PROGRAM FindBundlesFromDB EXTENDS SqldbReadWrite
VAR_INPUT
	id : STRING;
END_VAR
VAR_OUTPUT
	basicBundlesArr : ARRAY[0..20-1] OF BasicBundle;
END_VAR
VAR
	fbSQLCommand : FB_SQLCommandEvt(sNetID := '', tTimeout := T#5S);
	fbSQLDatabase : FB_SQLDatabaseEvt (sNetID := '', tTimeout := T#5S);
	fbSQLResult : FB_SQLResultEvt(sNetID:='', tTimeout:=T#5S);
	
	query : STRING(1000);
	//step : (RESET, CONNECT, IDLE, EXECUTE, LOAD_DATA, DISCONNECT);
END_VAR
VAR
	stringBuilder : StringBuilder;
	i : INT;
END_VAR

IF NOT ready THEN
	setup();
	RETURN;
END_IF

CASE step OF
	(*
	RESET:
		step := DISCONNECT;
		
	CONNECT:
		IF fbSQLDatabase.Connect(1) THEN
			IF NOT fbSqlDatabase.bError THEN
				step := IDLE;
			END_IF
		END_IF
	*)
	IDLE:
		IF fbSQLDatabase.CreateCmd(ADR(fbSQLCommand)) THEN
			step := EXECUTE;
		END_IF
	
	EXECUTE:
		createQuery();
		IF fbSQLCommand.ExecuteDataReturn(ADR(query), SIZEOF(query), ADR(fbSqlResult)) THEN
			step := IDLE;
		END_IF
	
	LOAD_DATA:
		(*
		fbSqlResult.Read(0, 1, ADR(existingID), SIZEOF(existingID), TRUE, FALSE);
		IF BundleData.id = existingID THEN
			bundleExists := TRUE;
		ELSE
			bundleExists := FALSE;
		END_IF
		IF fbSQLDatabase.Disconnect() THEN
			fbSqlResult.Release();
			checkExistingBundles := TRUE;
			dbCheckStep := CONNECT;
		END_IF
		*)
		
	DISCONNECT:
		IF fbSQLDatabase.Disconnect() THEN
			step := CONNECT;
		END_IF
END_CASE

METHOD PRIVATE createQuery : BOOL
IF id = '' THEN //FINISH WITH OTHER BASIC ATTRIBUTES
	CONCAT2(ADR(query), ADR('SELECT BundleID FROM "Bundle Data - Prototype"'), ADR(query), SIZEOF(query));
ELSE
	CONCAT2(ADR(query), ADR('SELECT BundleID FROM "Bundle Data - Prototype" WHERE BundleID = $''), ADR(query), SIZEOF(query));
	CONCAT2(ADR(query), ADR(id), ADR(query), SIZEOF(query));
	CONCAT2(ADR(query), ADR('$''), ADR(query), SIZEOF(query));
END_IF

createQuery := TRUE;
END_METHOD

METHOD queryBasicAttributes : BOOL
VAR_INPUT
END_VAR
END_METHOD

METHOD queryPackagingRecipe : BOOL
VAR_INPUT
	material : MaterialType;
END_VAR
VAR
	sMaterial : STRING;
END_VAR
sMaterial := TO_STRING(material);

IF i >= GVL.maxPairs THEN
	i := 0;
END_IF

sMaterial := stringBuilder
	.concatWith(
		'SELECT
		(position, top, sides, bottom, upperCorners, upperCorners_foldRatio, lowerCorners, lowerCorners_foldRatio)
		FROM ______ 
		WHERE (')
		
	.concatWith('bundleID = ')
	.concatWith('$'')
	.concatWith(TO_STRING(id))
	.concatWith('$'')
	
	.concatWith(' AND ')
	
	.concatWith('arrayIndex = ')
	.concatWith(TO_STRING(i))
	.concatWith(')')
	.getResult();
(*

FOR i:=0 TO 16 BY 1 DO


select (position, top, sides, bottom, upperCorners, upperCorners_foldRatio, lowerCorners, lowerCorners_foldRatio) from 
where (bundleID = bundle.id and arrayIndex = 1)

//copy the resulting cache into a bundle.<material>[i] (a PositionMaterial struct)
//do this for all material arrays


END_FORR

*)
END_METHOD

METHOD setup : BOOL
CASE step OF
	RESET:
		step := DISCONNECT;
		
	CONNECT:
		IF fbSQLDatabase.Connect(1) THEN
			IF NOT fbSqlDatabase.bError THEN
				step := IDLE;
				setup := TRUE;
			END_IF
		END_IF
		
	DISCONNECT:
		IF fbSQLDatabase.Disconnect() THEN
			step := CONNECT;
		END_IF
END_CASE
END_METHOD

END_PROGRAM

(* stored: Version 1.1.0.1, ProductVersion 3.1.4024.11
   POU FindBundlesFromDB: Id {75a3777c-6837-4547-91ca-cb43edd084bf}, SpecialFunc None
   Method createQuery: Id {efb6b343-7941-431a-a6cb-c4561387dac4}
   Method queryBasicAttributes: Id {91de8155-f84d-48ba-a38c-31179aab634d}
   Method queryPackagingRecipe: Id {71f08b57-21b8-4d7a-905d-a4f7abcc7830}
   Method setup: Id {2da3e218-e980-4fce-bd7a-62dcc22cc354} *)
